// TIA Portal V19 export
DATA_BLOCK "Config"   // DB31
// stored: Access Published, MemoryReserve 100, Namespace Unit2.EM3
   VAR
      em { ExternalWritable := 'False'} : "LAF_typeEmConfiguration";   // Configuration of EM Parameters
      axis { ExternalWritable := 'False'} : Array[1.._.U2EM3_NO_OF_AXES] of DB_ANY;   // Assign the axis of the EM
      cm6SlideCylinder { S7_SetPoint := 'True'} : "LBC_Simple_typeTwoWayActuatorConfiguration";
      cm7hookClawCylinder { S7_SetPoint := 'True'} : "LBC_Simple_typeTwoWayActuatorConfiguration";
      em3Parameters { S7_SetPoint := 'True'} : "LAF_typeConstraintWorkstationEm3Parameters";
   END_VAR
BEGIN
   em.referenceDesignator.parent := WSTRING#'U1';
   em.referenceDesignator.relative := WSTRING#'EM1';
   // em3Parameters.cm3Axis115.production.distanceList[0] : 低速小扭矩
   // em3Parameters.cm3Axis115.production.distanceList[1] : 高速大扭矩
   em3Parameters.cm3Axis115.production.distanceList[0..1].position := 0.0;
   em3Parameters.cm3Axis115.production.distanceList[0].velocity := 20.0;
   em3Parameters.cm3Axis115.production.distanceList[1].velocity := 50.0;
   em3Parameters.cm3Axis115.production.distanceList[0..1].acceleration := -1.0;
   em3Parameters.cm3Axis115.production.distanceList[0..1].deceleration := -1.0;
   em3Parameters.cm3Axis115.production.distanceList[0].torqueLimit := 1.0;
   em3Parameters.cm3Axis115.production.distanceList[1].torqueLimit := 2.0;
   // em3Parameters.cm4Axis116.production.distanceList[0] : 低速小扭矩
   // em3Parameters.cm4Axis116.production.distanceList[1] : 高速大扭矩
   em3Parameters.cm4Axis116.production.distanceList[0].velocity := 20.0;
   em3Parameters.cm4Axis116.production.distanceList[1].velocity := 50.0;
   em3Parameters.cm4Axis116.production.distanceList[0].torqueLimit := 1.0;
   em3Parameters.cm4Axis116.production.distanceList[1].torqueLimit := 2.0;
END_DATA_BLOCK
